TYPE MastLightReq :
STRUCT

RedReq: BOOL;
RedFlashReq: BOOL;
YelReq: BOOL;
YelFlashReq: BOOL;
GrnReq: BOOL;
GrnFlashReq: BOOL;
HornReq: BOOL;	

END_STRUCT
END_TYPE

(* stored: Version 1.1.0.1, ProductVersion 3.1.4024.6
   DUT MastLightReq: Id {8de2fa03-a003-4138-875e-31325c67c043} *)
